// TIA Portal V17 export
// export: Created 2024-08-09T12:53:10.119461Z, ExportSetting WithDefaults, DisplayName Totally Integrated Automation Portal, DisplayVersion V17 Update 7, DisplayName TIA Portal Openness, DisplayVersion V17 Update 7, DisplayName TIA Portal Version Control Interface, DisplayVersion V17, DisplayName STEP 7 Professional, DisplayVersion V17 Update 7, DisplayName STEP 7 Safety, DisplayVersion V17 Update 6, DisplayName WinCC Professional, DisplayVersion V17 Update 7
VAR_GLOBAL   // PLC tag table "Taches"
END_VAR
VAR_GLOBAL CONSTANT   // user constants
   TAC_BP1 : SInt := 0;   // Numero tache benne BP1
   TAC_BP2 : SInt := 1;   // Numero tache benne BP2
   TAC_CIRREMP_BR1 : SInt := 10;   // Numero tache circuit transfet remplissage boisseaux sur broyeur1
   TAC_CIRREMP_BR2 : SInt := 11;   // Numero tache circuit transfet remplissage boisseaux sur broyeur2
   TAC_BR1 : SInt := 12;   // Numero tache broyeur BR1
   TAC_BR2 : SInt := 13;   // Numero tache broyeur BR2
   TAC_TREMSS_BR1 : SInt := 14;   // Numero tache tremie sous broyeur BR1
   TAC_TREMSS_BR2 : SInt := 15;   // Numero tache tremie sous broyeur BR2
   TAC_TREMSR_BR1 : SInt := 16;   // Numero tache tremie sur broyeur BR1
   TAC_TREMSR_BR2 : SInt := 17;   // Numero tache tremie sur broyeur BR2
   TAC_CIRREMP_MLG1 : SInt := 18;   // Numero tache circuit transfet remplissage boisseaux sur melangeuse1
   TAC_CIRREMP_MLG2 : SInt := 19;   // Numero tache circuit transfet remplissage boisseaux sur melangeuse2
   TAC_BP3 : SInt := 2;   // Numero tache benne BP3
   TAC_TREMSR_MLG1 : SInt := 20;   // Numero tache tremie sur melangeuse1
   TAC_MELANG1 : SInt := 21;   // Numero tache melangeuse1
   TAC_TREMSS_MLG1 : SInt := 22;   // Numero tache tremie sous melangeuse1
   TAC_LIQ1_MLG1 : SInt := 23;   // Numero tache Liquide1 melangeuse1
   TAC_LIQ2_MLG1 : SInt := 24;   // Numero tache Liquide2 melangeuse1
   TAC_LIQ3_MLG1 : SInt := 25;   // Numero tache Liquide3 melangeuse1
   TAC_DEROUT_EXP : SInt := 26;   // Numero tache deroutage expedition
   TAC_LANC_EXP : SInt := 27;   // Numero tache lancement expedition
   TAC_EXP1 : SInt := 28;   // Numero tache expedition1
   TAC_EXP2 : SInt := 29;   // Numero tache expedition2
   TAC_BP4 : SInt := 3;   // Numero tache benne BP4
   TAC_CIRSS_BP1 : SInt := 30;   // Numero tache circuit transfert sous BP1
   TAC_VS_MLG1 : SInt := 31;   // Numero tache Verse Sac Melangeuse1
   TAC_VS_MLG2 : SInt := 32;   // Numero tache Verse Sac Melangeuse2
   TAC_MELANG2 : SInt := 33;   // Numero tache circuit transfet remplissage boisseaux sur melangeuse2
   TAC_TREMSR_MLG2 : SInt := 34;   // Numero tache tremie sur melangeuse2
   TAC_TREMSS_MLG2 : SInt := 35;   // Numero tache tremie sous melangeuse2
   TAC_LIQ4_MLG1 : SInt := 36;   // Numero tache Liquide4 melangeuse1
   TAC_LIQ5_MLG1 : SInt := 37;   // Numero tache Liquide5 melangeuse1
   TAC_LIQ1_MLG2 : SInt := 38;   // Numero tache Liquide1 melangeuse2
   TAC_LIQ2_MLG2 : SInt := 39;   // Numero tache Liquide2 melangeuse2
   TAC_BP5 : SInt := 4;   // Numero tache benne BP5
   TAC_LIQ3_MLG2 : SInt := 40;   // Numero tache Liquide3 melangeuse2
   TAC_LIQ4_MLG2 : SInt := 41;   // Numero tache Liquide4 melangeuse2
   TAC_LIQ5_MLG2 : SInt := 42;   // Numero tache Liquide5 melangeuse2
   TAC_TREMSS_BP1 : SInt := 5;   // Numero tache tremie sous BP1
   TAC_TREMSS_BP2 : SInt := 6;   // Numero tache tremie sous BP2
   TAC_TREMSS_BP3 : SInt := 7;   // Numero tache tremie sous BP3
   TAC_TREMSS_BP4 : SInt := 8;   // Numero tache tremie sous BP4
   TAC_TREMSS_BP5 : SInt := 9;   // Numero tache tremie sous BP5
   TAC_REC1 : SInt := 43;   // Numero tache reception 1
   TAC_REC2 : SInt := 44;   // Numero tache reception 2
   TAC_REC3 : SInt := 45;   // Numero tache reception 3
   TAC_REC4 : SInt := 46;   // Numero tache reception 4
   TAC_TRANSF : SInt := 47;   // Numero tache TRANSFERT
   TAC_GTOUR : SInt := 48;   // Numero tache gestion tournee
   TAC_PONT1 : SInt := 49;   // Numero tache chargement pont
   TAC_VIDCEL : SInt := 50;   // Numero tache VIDANGE CELLULE
END_VAR
